{region '#Template'}
	{attribute 'Category' := 'AC'}
	{attribute 'Version' := '0.0.1.0'}
	{attribute 'Tags' := 'AC, Aggregates, Cooler, Temperature, Controller'}
	{attribute 'Description' := 'Kühler Zuluft Regler Temperatur	// Cooler Supply air controller temperature'}
{endregion}
FUNCTION_BLOCK FB_BA_AC_ColTSuACtrl EXTENDS FB_BA_View
VAR_INPUT
	bEn						: BOOL;
	fSpTSuA					: REAL;
	fTSuA					: REAL;
	bSync					: BOOL;
	fSync					: REAL;
END_VAR
VAR_OUTPUT
	fY              		: REAL;
	bIsActive				: BOOL;	//	active sequence controller
	bOpState				: BOOL;	//	Release sequence link, sequence control is active	
END_VAR
VAR_INPUT CONSTANT
	Ctrl					: FB_BA_Loop;
END_VAR

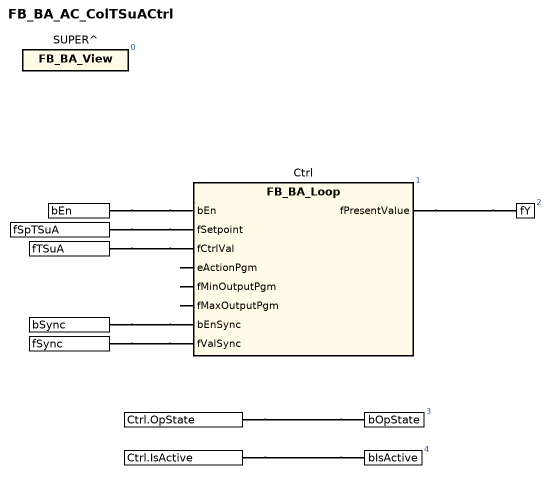
SUPER^(); // FB_BA_View
Ctrl(bEn := bEn, fSetpoint := fSpTSuA, fCtrlVal := fTSuA, bEnSync := bSync, fValSync := fSync); // FB_BA_Loop
fY := Ctrl.fPresentValue;
bOpState := Ctrl.OpState;
bIsActive := Ctrl.IsActive;

METHOD FB_init : BOOL
VAR_INPUT
	bInitRetains : BOOL; // if TRUE, the retain variables are initialized (warm start / cold start)
	bInCopyCode : BOOL;  // if TRUE, the instance afterwards gets moved into the copy code (online change)
END_VAR
Ctrl.iParent						:= THIS^;
Ctrl.iLabel							:= LblCmpAC.Cooler_TSuACtrl_Ctrl; 
Ctrl.sObjectName					:= '{Idx=01}';
Ctrl.eOpMode						:= BA2_Param.nLoop_DefOpMode;								 	 										 
Ctrl.eOutputUnit					:= E_BA_Unit.eOther_Percent;
Ctrl.eActionRm						:= E_BA_Action.eDirect;
Ctrl.fProportionalConstant			:= 3;
Ctrl.fIntegralConstant				:= 180;
Ctrl.fDerivativeConstant			:= 0;
Ctrl.fMaxOutputRm 					:= 100;
Ctrl.fMinOutputRm					:= 0;
Ctrl.fCOVIncrement					:= 0;
Ctrl.nDampConstant					:= 0;
Ctrl.fNeutralZone					:= 0;
Ctrl.stStepDelay.nDown				:= 0;
Ctrl.stStepDelay.nUp				:= 0;
END_METHOD

END_FUNCTION_BLOCK

(* stored: Version 1.1.0.1, ProductVersion 3.1.4024.6
   POU FB_BA_AC_ColTSuACtrl: Id {b00970de-a0ac-486b-8361-2d5585e2b95f}, SpecialFunc None
   Method FB_init: Id {d7d20e92-4553-4504-9685-492b4e0687c5} *)
